(* Schneider Machine Expert - Basic project share resources, file version 2.7.0.0 *)
(* ProjectInformations: Name=Nuevo proyecto *)

HARDWARE
  Cpu 0: TM221C16R
  ModuleExtensionObject 0: TM3AQ2/G
  EthernetConfiguration: NetworkName=M221, IpAllocationMode=FixedAddress, IpAddress=0.0.0.0, SubnetMask=0.0.0.0
  SerialLineConfiguration: Baud=Baud19200, Parity=ParityEven, DataBits=DataBits8, StopBits=StopBits1, PhysicalMedium=PhysicalMediumRs485, TransmissionMode=TransmissionModeModbusRtu, SlaveId=1, Addressing=SlaveAddressing
  MastTask: UsePeriodScanMode=false, PeriodScan=100
  FastTask: Period=255
  CpuBehavior: StartingMode=StartAsPreviousState, AutoSaveRamOnEeprom=true, WatchdogPeriod=250

SYMBOLS  (address, symbol, comment, settings)
  %M0       AT_ENTRY_1
  %M1       AT_ENTRY_2
  %M2       AT_TRANSFER_1
  %M3       AT_TRANSFER_2
  %M4       AT_EXIT
  %M5       BUTTON_START
  %M6       BUTTON_RESET
  %M7       BUTTON_STOP
  %M8       BUTTON_EMERGENCY_STOP
  %M9       BUTTON_AUTO
  %M11      CONVEYOR_1
  %M12      LOAD_1
  %M15      TRANSFER_LEFT_1
  %M16      CONVEYOR_2
  %M17      LOAD_2
  %M20      TRANSFER_LEFT_2
  %M21      EXIT_CONVEYOR
  %M22      START_LIGHT
  %M23      RESET_LIGHT
  %M24      STOP_LIGHT
  %M100     AUTO_ACTIVE
  %X1       ESTADO_1
  %X2       ESTADO_2
  %X3       ESTADO_3
  %X4       ESTADO_4
  %X5       ESTADO_5
  %X6       ESTADO_6
  %X7       ESTADO_7
  %X8       ESTADO_8
  %X9       ESTADO_9
  %X10      ESTADO_10
  %X11      ESTADO_11
  %TM0      STATE_4_TIMER  [Type=TOF, Preset=65, Base=OneHundredMilliSeconds]
  %TM1      STATE_11_TIMER  [Type=TOF, Preset=65, Base=OneHundredMilliSeconds]

GRAFCET Share resource
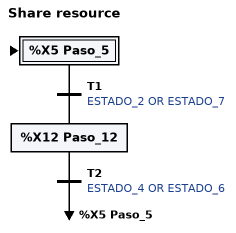
  INITIAL_STEP %X5  (* Paso_5 *)
  STEP %X12  (* Paso_12 *)
  TRANSITION T1 FROM %X5 TO %X12 := ESTADO_2 OR ESTADO_7;
  TRANSITION T2 FROM %X12 TO %X5 := ESTADO_4 OR ESTADO_6;

GRAFCET Grafcet 2
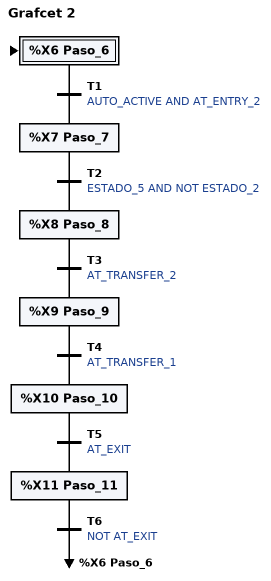
  INITIAL_STEP %X6  (* Paso_6 *)
  STEP %X7  (* Paso_7 *)
  STEP %X8  (* Paso_8 *)
  STEP %X9  (* Paso_9 *)
  STEP %X10  (* Paso_10 *)
  STEP %X11  (* Paso_11 *)
  TRANSITION T1 FROM %X6 TO %X7 := AUTO_ACTIVE AND AT_ENTRY_2;
  TRANSITION T2 FROM %X7 TO %X8 := ESTADO_5 AND NOT ESTADO_2;
  TRANSITION T3 FROM %X8 TO %X9 := AT_TRANSFER_2;
  TRANSITION T4 FROM %X9 TO %X10 := AT_TRANSFER_1;
  TRANSITION T5 FROM %X10 TO %X11 := AT_EXIT;
  TRANSITION T6 FROM %X11 TO %X6 := NOT AT_EXIT;

GRAFCET Grafcet 1
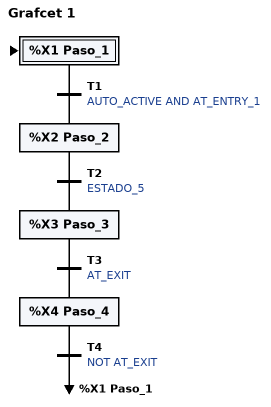
  INITIAL_STEP %X1  (* Paso_1 *)
  STEP %X2  (* Paso_2 *)
  STEP %X3  (* Paso_3 *)
  STEP %X4  (* Paso_4 *)
  TRANSITION T1 FROM %X1 TO %X2 := AUTO_ACTIVE AND AT_ENTRY_1;
  TRANSITION T2 FROM %X2 TO %X3 := ESTADO_5;
  TRANSITION T3 FROM %X3 TO %X4 := AT_EXIT;
  TRANSITION T4 FROM %X4 TO %X1 := NOT AT_EXIT;

POU Buttons
  (* SectionNumber=1 *)

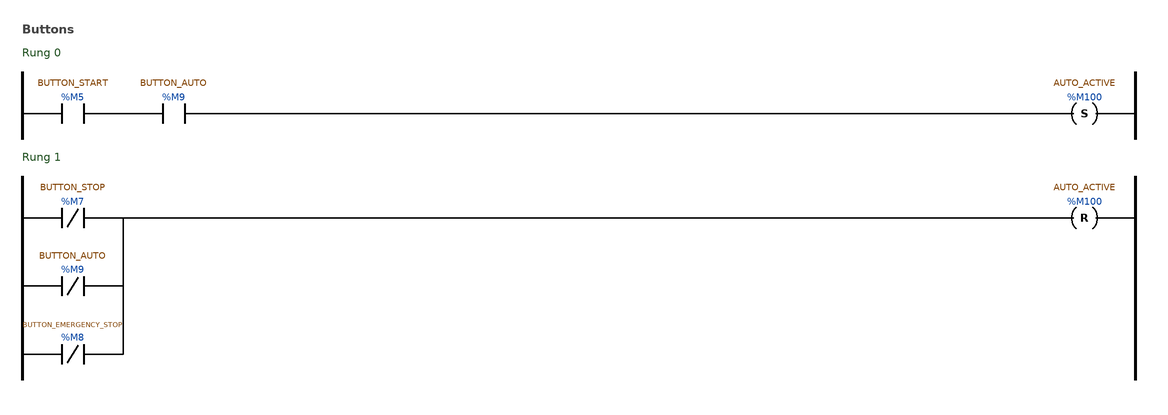

// Rung 0
  LD %M5                  (* BUTTON_START *)
  AND %M9                 (* BUTTON_AUTO *)
  S %M100                 (* AUTO_ACTIVE *)
  // as ST:
  //   IF BUTTON_START AND BUTTON_AUTO THEN AUTO_ACTIVE := TRUE; END_IF;

// Rung 1
  LDN %M7                 (* BUTTON_STOP *)
  ORN %M9                 (* BUTTON_AUTO *)
  ORN %M8                 (* BUTTON_EMERGENCY_STOP *)
  R %M100                 (* AUTO_ACTIVE *)
  // as ST:
  //   IF NOT BUTTON_STOP OR NOT BUTTON_AUTO OR NOT BUTTON_EMERGENCY_STOP THEN AUTO_ACTIVE := FALSE; END_IF;

TRANSITION T1 (%X5 -> %X12) 
  (* SectionNumber=0 *)

// Rung 2: Tr1
  LD %X2                  (* ESTADO_2 *)
  OR %X7                  (* ESTADO_7 *)
  ENDT
  // as ST:
  //   TRANSITION := ESTADO_2 OR ESTADO_7;

TRANSITION T2 (%X12 -> %X5) 
  (* SectionNumber=0 *)

// Rung 3: Tr2
  LD %X4                  (* ESTADO_4 *)
  OR %X6                  (* ESTADO_6 *)
  ENDT
  // as ST:
  //   TRANSITION := ESTADO_4 OR ESTADO_6;

TRANSITION T1 (%X6 -> %X7) 
  (* SectionNumber=0 *)

// Rung 4: Tr1
  LD %M100                (* AUTO_ACTIVE *)
  AND %M1                 (* AT_ENTRY_2 *)
  ENDT
  // as ST:
  //   TRANSITION := AUTO_ACTIVE AND AT_ENTRY_2;

TRANSITION T2 (%X7 -> %X8) 
  (* SectionNumber=0 *)

// Rung 5: Tr2
  LD %X5                  (* ESTADO_5 *)
  ANDN %X2                (* ESTADO_2 *)
  ENDT
  // as ST:
  //   TRANSITION := ESTADO_5 AND NOT ESTADO_2;

TRANSITION T3 (%X8 -> %X9) 
  (* SectionNumber=0 *)

// Rung 6: Tr3
  LD %M3                  (* AT_TRANSFER_2 *)
  ENDT
  // as ST:
  //   TRANSITION := AT_TRANSFER_2;

TRANSITION T4 (%X9 -> %X10) 
  (* SectionNumber=0 *)

// Rung 7: Tr4
  LD %M2                  (* AT_TRANSFER_1 *)
  ENDT
  // as ST:
  //   TRANSITION := AT_TRANSFER_1;

TRANSITION T5 (%X10 -> %X11) 
  (* SectionNumber=0 *)

// Rung 8: Tr5
  LD %M4                  (* AT_EXIT *)
  ENDT
  // as ST:
  //   TRANSITION := AT_EXIT;

TRANSITION T6 (%X11 -> %X6) 
  (* SectionNumber=0 *)

// Rung 9: Tr6
  LDN %M4                 (* AT_EXIT *)
  ENDT
  // as ST:
  //   TRANSITION := NOT AT_EXIT;

TRANSITION T1 (%X1 -> %X2) 
  (* SectionNumber=0 *)

// Rung 10: Tr1
  LD %M100                (* AUTO_ACTIVE *)
  AND %M0                 (* AT_ENTRY_1 *)
  ENDT
  // as ST:
  //   TRANSITION := AUTO_ACTIVE AND AT_ENTRY_1;

TRANSITION T2 (%X2 -> %X3) 
  (* SectionNumber=0 *)

// Rung 11: Tr2
  LD %X5                  (* ESTADO_5 *)
  ENDT
  // as ST:
  //   TRANSITION := ESTADO_5;

TRANSITION T3 (%X3 -> %X4) 
  (* SectionNumber=0 *)

// Rung 12: Tr3
  LD %M4                  (* AT_EXIT *)
  ENDT
  // as ST:
  //   TRANSITION := AT_EXIT;

TRANSITION T4 (%X4 -> %X1) 
  (* SectionNumber=0 *)

// Rung 13: Tr10
  LDN %M4                 (* AT_EXIT *)
  ENDT
  // as ST:
  //   TRANSITION := NOT AT_EXIT;

POU Lights
  (* SectionNumber=15 *)

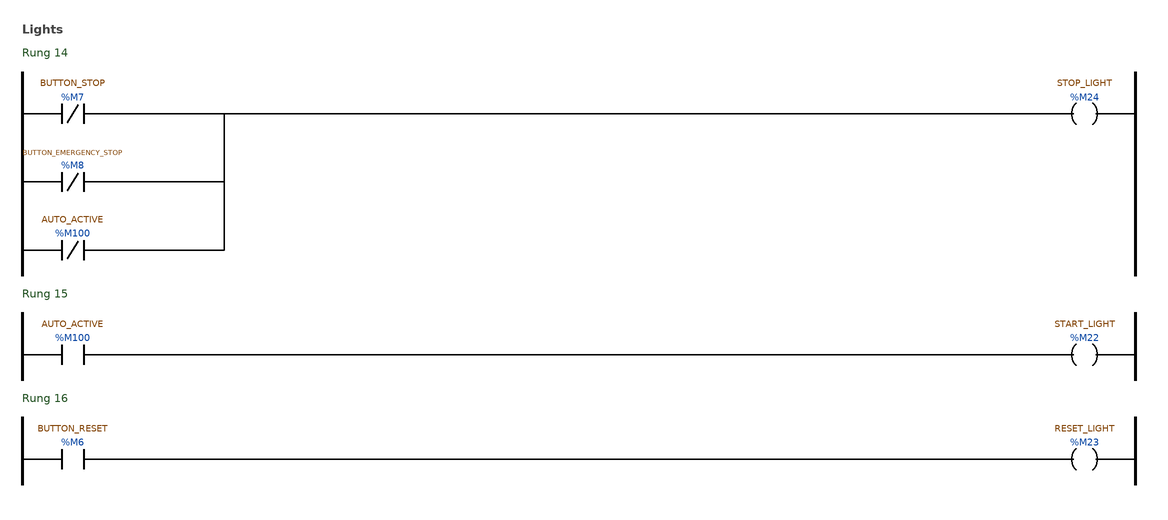

// Rung 14
  LDN %M7                 (* BUTTON_STOP *)
  ORN %M8                 (* BUTTON_EMERGENCY_STOP *)
  ORN %M100               (* AUTO_ACTIVE *)
  ST %M24                 (* STOP_LIGHT *)
  // as ST:
  //   STOP_LIGHT := NOT BUTTON_STOP OR NOT BUTTON_EMERGENCY_STOP OR NOT AUTO_ACTIVE;

// Rung 15
  LD %M100                (* AUTO_ACTIVE *)
  ST %M22                 (* START_LIGHT *)
  // as ST:
  //   START_LIGHT := AUTO_ACTIVE;

// Rung 16
  LD %M6                  (* BUTTON_RESET *)
  ST %M23                 (* RESET_LIGHT *)
  // as ST:
  //   RESET_LIGHT := BUTTON_RESET;

POU Actions
  (* SectionNumber=16 *)

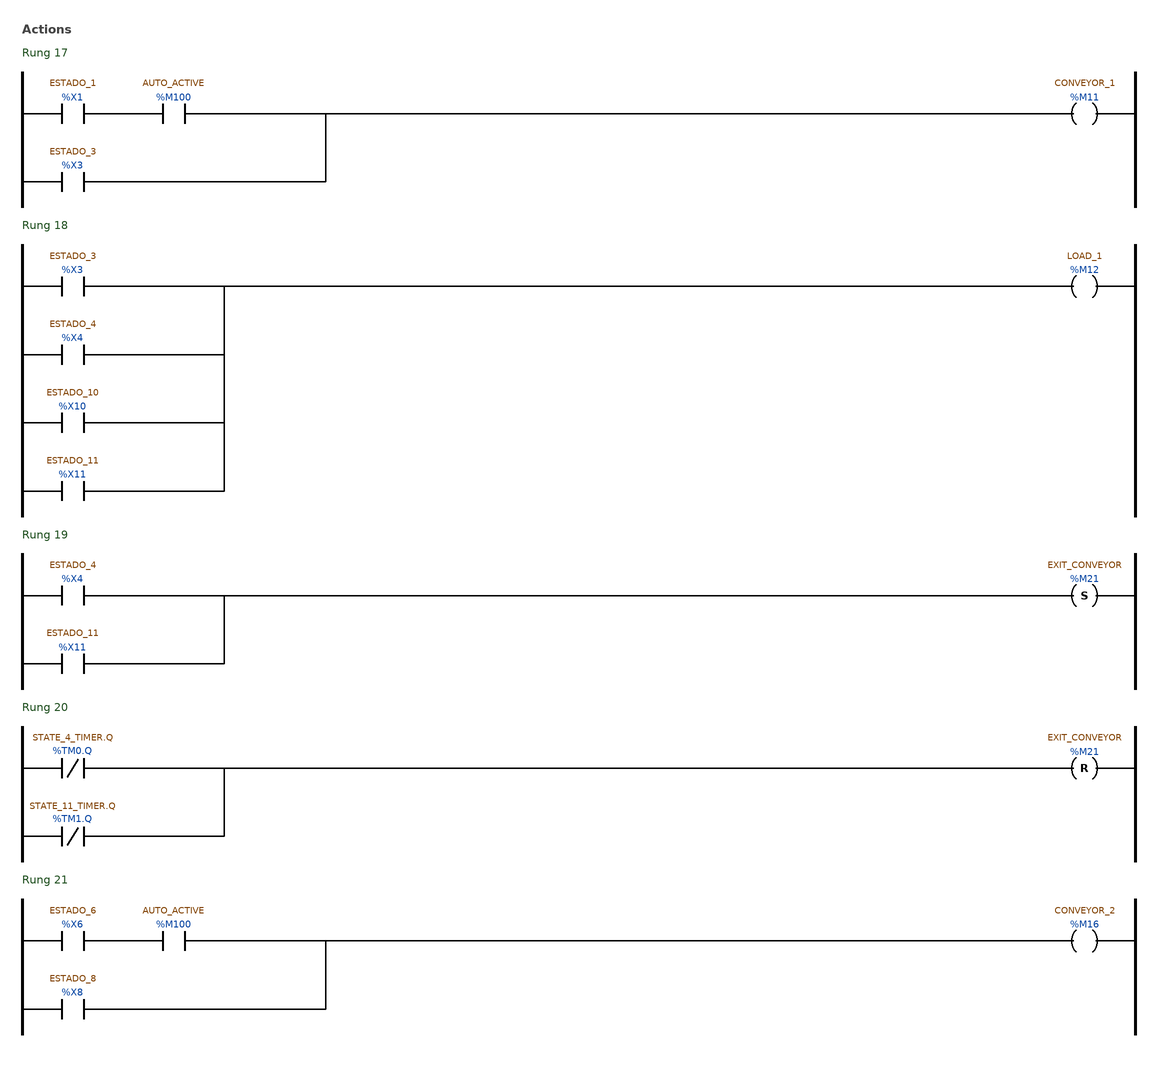

// Rung 17
  LD %X1                  (* ESTADO_1 *)
  AND %M100               (* AUTO_ACTIVE *)
  OR %X3                  (* ESTADO_3 *)
  ST %M11                 (* CONVEYOR_1 *)
  // as ST:
  //   CONVEYOR_1 := ESTADO_1 AND AUTO_ACTIVE OR ESTADO_3;

// Rung 18
  LD %X3                  (* ESTADO_3 *)
  OR %X4                  (* ESTADO_4 *)
  OR %X10                 (* ESTADO_10 *)
  OR %X11                 (* ESTADO_11 *)
  ST %M12                 (* LOAD_1 *)
  // as ST:
  //   LOAD_1 := ESTADO_3 OR ESTADO_4 OR ESTADO_10 OR ESTADO_11;

// Rung 19
  LD %X4                  (* ESTADO_4 *)
  OR %X11                 (* ESTADO_11 *)
  S %M21                  (* EXIT_CONVEYOR *)
  // as ST:
  //   IF ESTADO_4 OR ESTADO_11 THEN EXIT_CONVEYOR := TRUE; END_IF;

// Rung 20
  LDN %TM0.Q              (* STATE_4_TIMER *)
  ORN %TM1.Q              (* STATE_11_TIMER *)
  R %M21                  (* EXIT_CONVEYOR *)
  // as ST:
  //   IF NOT STATE_4_TIMER.Q OR NOT STATE_11_TIMER.Q THEN EXIT_CONVEYOR := FALSE; END_IF;

// Rung 21
  LD %X6                  (* ESTADO_6 *)
  AND %M100               (* AUTO_ACTIVE *)
  OR %X8                  (* ESTADO_8 *)
  ST %M16                 (* CONVEYOR_2 *)
  // as ST:
  //   CONVEYOR_2 := ESTADO_6 AND AUTO_ACTIVE OR ESTADO_8;

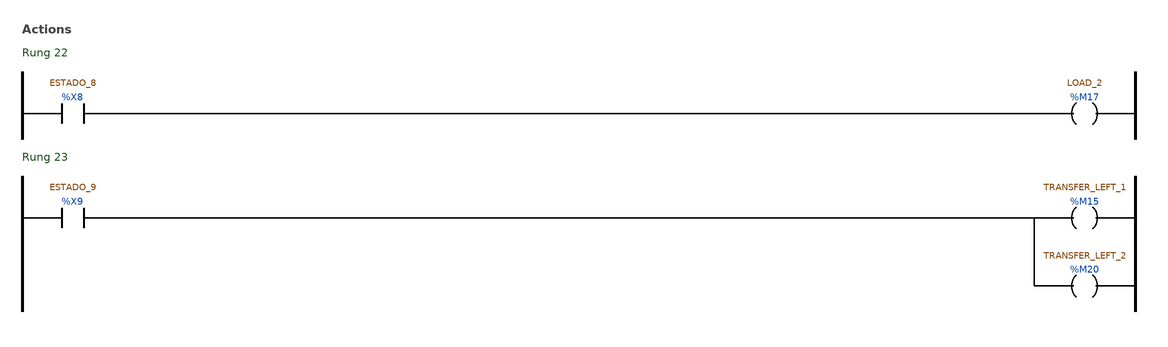

// Rung 22
  LD %X8                  (* ESTADO_8 *)
  ST %M17                 (* LOAD_2 *)
  // as ST:
  //   LOAD_2 := ESTADO_8;

// Rung 23
  LD %X9                  (* ESTADO_9 *)
  ST %M15                 (* TRANSFER_LEFT_1 *)
  ST %M20                 (* TRANSFER_LEFT_2 *)
  // as ST:
  //   TRANSFER_LEFT_1 := ESTADO_9;
  //   TRANSFER_LEFT_2 := ESTADO_9;

POU Timers and counters
  (* SectionNumber=17 *)

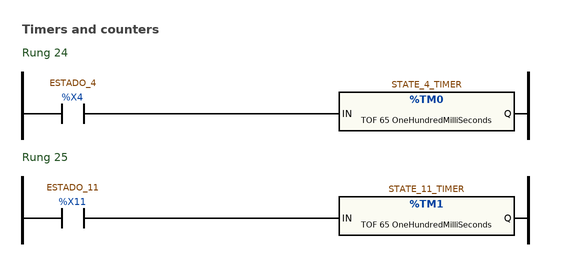

// Rung 24
  BLK %TM0                (* STATE_4_TIMER *)
  LD %X4                  (* ESTADO_4 *)
  IN
  END_BLK
  // as ST:
  //   STATE_4_TIMER(IN := ESTADO_4);

// Rung 25
  BLK %TM1                (* STATE_11_TIMER *)
  LD %X11                 (* ESTADO_11 *)
  IN
  END_BLK
  // as ST:
  //   STATE_11_TIMER(IN := ESTADO_11);
